Universal Robots PolyScope program: Lab_exe_5_1_98.urp

Program Lab_exe_5_1_98 (createdIn=3.2.19293 lastSavedIn=3.2.19293 directory=/programs installation=default robotSerialNumber=2015351391)
Calibrated DH parameters: a=[0.000352, -0.161198, -0.373486, 0.00005, 0.000049, 0]; d=[0.089268, 352.477598, -320.08558, -32.281492, 0.094939, 0.082518]; alpha=[1.570728, 0.001116, -0.003686, 1.571189, -1.570572, 0]; deltaTheta=[-0.000012, 1.181849, -1.491165, 0.309495, -0.000007, 0.000025]
Robot Program (runOnlyOnce=true motionType=MoveJ speed=1.047198 acceleration=1.396263 recalculateMotions=false)
  Loop Counting (count=5) loopVariable(name=循环_1)
    Call SubP_lamp_flash
SubProgram -> SubP_lamp_flash
SubProgram SubP_lamp_flash (keepSynchronizedWithDisk=false trackProgramExecution=false) programFile=/programs/lamp_flash.urp
  Set DigitalOutput pin=Lamp; digitalValue=1
  Wait Sleep waitTime=0.5
  Set DigitalOutput pin=Lamp; digitalValue=0
  Wait Sleep waitTime=0.5
